FUNCTION_BLOCK FB_Siemens
   VAR_INPUT 
      input : Bool;
      inputreal : Real;
   END_VAR

   VAR_OUTPUT 
      outputreal : Real;
   END_VAR


          	IF #input = TRUE THEN
	    #outputreal := #inputreal;
	END_IF;
	//oder
	IF #input = FALSE THEN
	    #outputreal := #inputreal / 2;
	END_IF;

END_FUNCTION_BLOCK

(* stored: Version 1.1.0.1, ProductVersion 3.1.4024.9
   POU FB_Siemens: Id {1c07b5fc-28d6-44e5-8f78-58efd977b308}, SpecialFunc None *)
